Staubli VAL3: getPalletList.pgx

program getPalletList()
begin
  //
  // INIT
  //
  libList(saveData:sPathTraj+"PALLET",sPalletName)
end
